PROGRAM pouMachine
VAR
	pnuOn: FB_Motion1way;
	isAirSwitchOn: BOOL;
	tAllPowerOn: BOOL;
	tAnyPowerOn: BOOL;
	tGate1AccessReq: BOOL;
	tGate2AccessReq: BOOL;
	FB_CheckAnyMode_0: FB_CheckAnyMode;
	tWaitMsgXICAdv: BOOL;
	tAnyManualReq: BOOL;
	tAnyAutoReq: BOOL;
END_VAR
VAR // added by the converter: edge detectors and wires of the graphical bodies
    _w1 : BOOL;
END_VAR

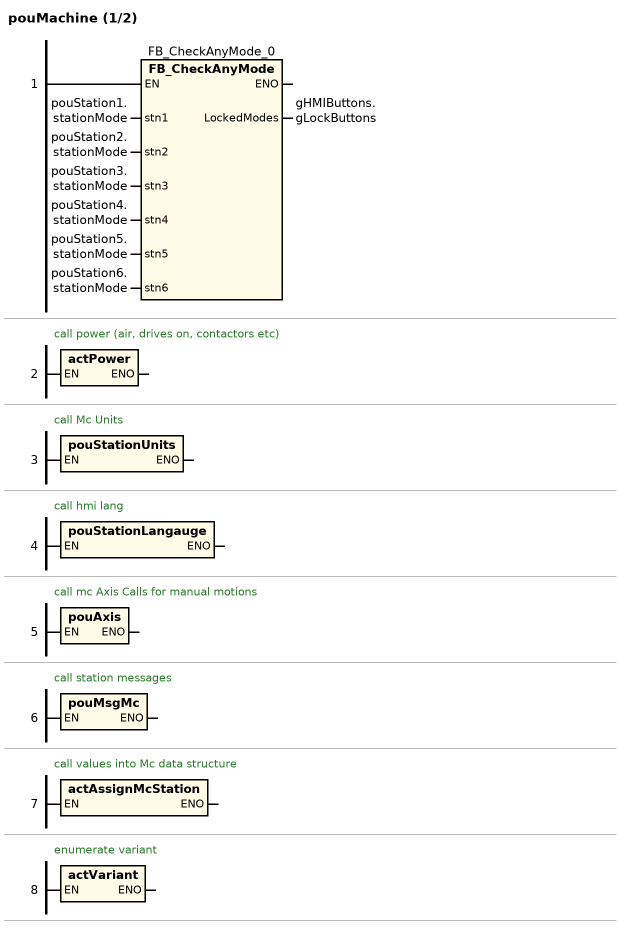
// NETWORK 1
FB_CheckAnyMode_0(
    stn1 := pouStation1.stationMode,
    stn2 := pouStation2.stationMode,
    stn3 := pouStation3.stationMode,
    stn4 := pouStation4.stationMode,
    stn5 := pouStation5.stationMode,
    stn6 := pouStation6.stationMode,
    LockedModes => gHMIButtons.gLockButtons); // FB_CheckAnyMode

// NETWORK 2
// call power (air, drives on, contactors etc)
actPower();

// NETWORK 3
// call Mc Units
pouStationUnits();

// NETWORK 4
// call hmi lang
pouStationLangauge();

// NETWORK 5
// call mc Axis Calls for manual motions
pouAxis();

// NETWORK 6
// call station messages
pouMsgMc();

// NETWORK 7
// call values into Mc data structure
actAssignMcStation();

// NETWORK 8
// enumerate variant
actVariant();

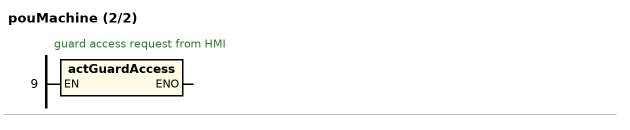
// NETWORK 9
// guard access request from HMI
actGuardAccess();

ACTION actAssignMcStation:
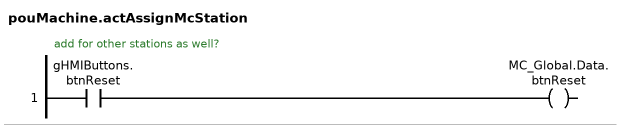
// NETWORK 1
// add for other stations as well?
MC_Global.Data.btnReset := gHMIButtons.btnReset;
END_ACTION

ACTION actGuardAccess:
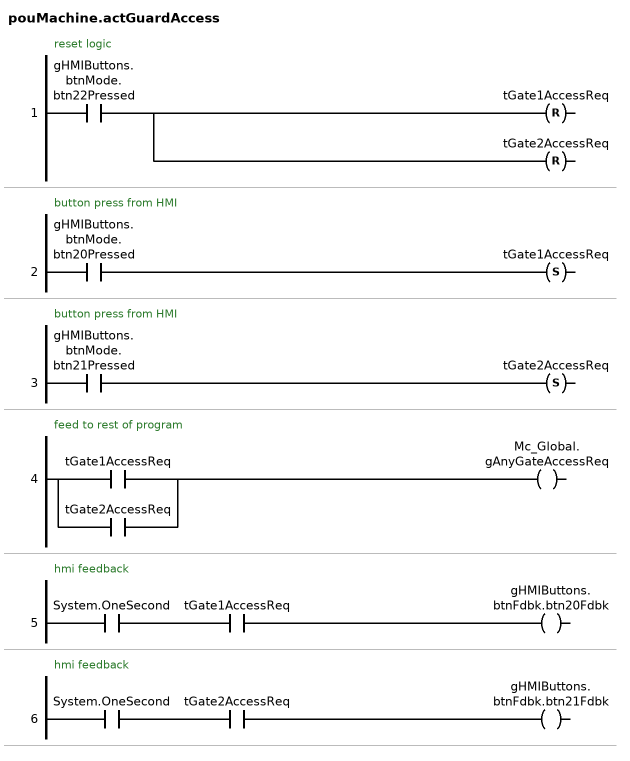
// NETWORK 1
// reset logic
tGate1AccessReq R= gHMIButtons.btnMode.btn22Pressed;
tGate2AccessReq R= gHMIButtons.btnMode.btn22Pressed;

// NETWORK 2
// button press from HMI
tGate1AccessReq S= gHMIButtons.btnMode.btn20Pressed;

// NETWORK 3
// button press from HMI
tGate2AccessReq S= gHMIButtons.btnMode.btn21Pressed;

// NETWORK 4
// feed to rest of program
Mc_Global.gAnyGateAccessReq := tGate1AccessReq OR tGate2AccessReq;

// NETWORK 5
// hmi feedback
gHMIButtons.btnFdbk.btn20Fdbk := System.OneSecond AND tGate1AccessReq;

// NETWORK 6
// hmi feedback
gHMIButtons.btnFdbk.btn21Fdbk := System.OneSecond AND tGate2AccessReq;
END_ACTION

ACTION actPower:
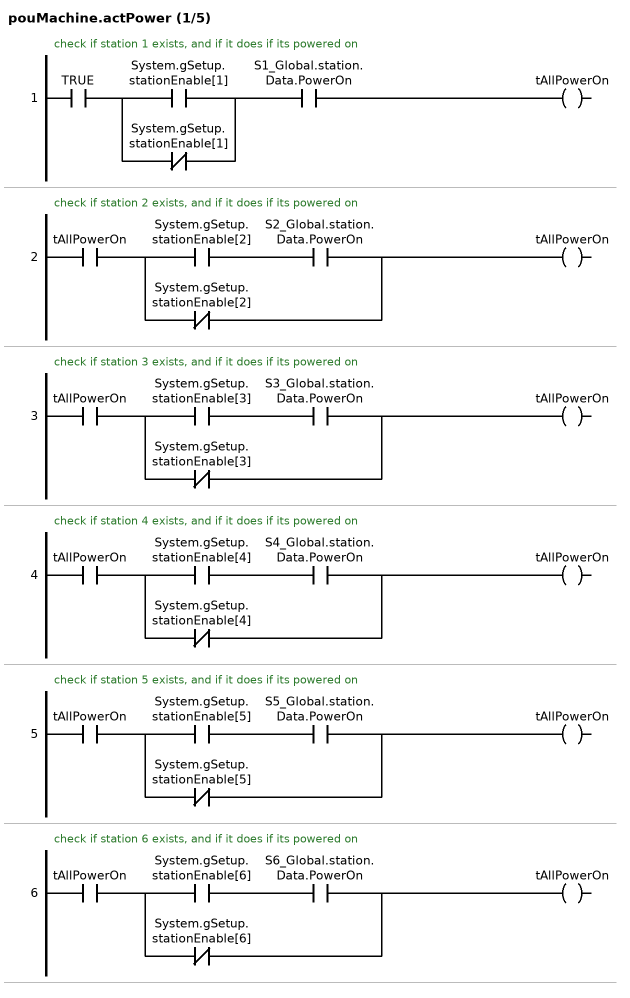
// NETWORK 1
// check if station 1 exists, and if it does if its powered on
tAllPowerOn := TRUE AND (System.gSetup.stationEnable[1] OR NOT System.gSetup.stationEnable[1]) AND S1_Global.station.Data.PowerOn;

// NETWORK 2
// check if station 2 exists, and if it does if its powered on
tAllPowerOn := tAllPowerOn AND (System.gSetup.stationEnable[2] AND S2_Global.station.Data.PowerOn OR NOT System.gSetup.stationEnable[2]);

// NETWORK 3
// check if station 3 exists, and if it does if its powered on
tAllPowerOn := tAllPowerOn AND (System.gSetup.stationEnable[3] AND S3_Global.station.Data.PowerOn OR NOT System.gSetup.stationEnable[3]);

// NETWORK 4
// check if station 4 exists, and if it does if its powered on
tAllPowerOn := tAllPowerOn AND (System.gSetup.stationEnable[4] AND S4_Global.station.Data.PowerOn OR NOT System.gSetup.stationEnable[4]);

// NETWORK 5
// check if station 5 exists, and if it does if its powered on
tAllPowerOn := tAllPowerOn AND (System.gSetup.stationEnable[5] AND S5_Global.station.Data.PowerOn OR NOT System.gSetup.stationEnable[5]);

// NETWORK 6
// check if station 6 exists, and if it does if its powered on
tAllPowerOn := tAllPowerOn AND (System.gSetup.stationEnable[6] AND S6_Global.station.Data.PowerOn OR NOT System.gSetup.stationEnable[6]);

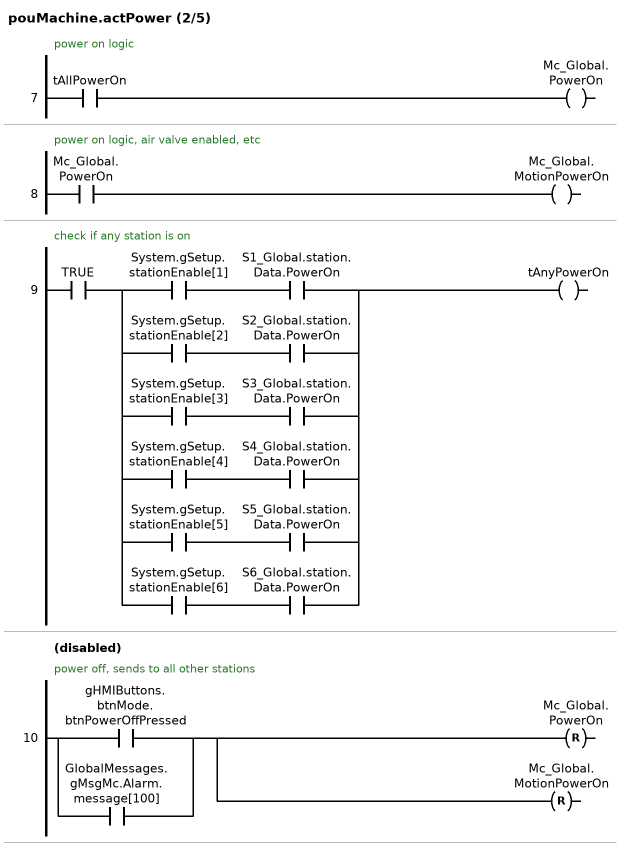
// NETWORK 7
// power on logic
Mc_Global.PowerOn := tAllPowerOn;

// NETWORK 8
// power on logic, air valve enabled, etc
Mc_Global.MotionPowerOn := Mc_Global.PowerOn;

// NETWORK 9
// check if any station is on
tAnyPowerOn := TRUE AND (System.gSetup.stationEnable[1] AND S1_Global.station.Data.PowerOn OR System.gSetup.stationEnable[2] AND S2_Global.station.Data.PowerOn OR System.gSetup.stationEnable[3] AND S3_Global.station.Data.PowerOn OR System.gSetup.stationEnable[4] AND S4_Global.station.Data.PowerOn OR System.gSetup.stationEnable[5] AND S5_Global.station.Data.PowerOn OR System.gSetup.stationEnable[6] AND S6_Global.station.Data.PowerOn);

// NETWORK 10 (disabled)
// power off, sends to all other stations
// _w1 := gHMIButtons.btnMode.btnPowerOffPressed OR GlobalMessages.gMsgMc.Alarm.message[100];
// Mc_Global.PowerOn R= _w1;
// Mc_Global.MotionPowerOn R= _w1;

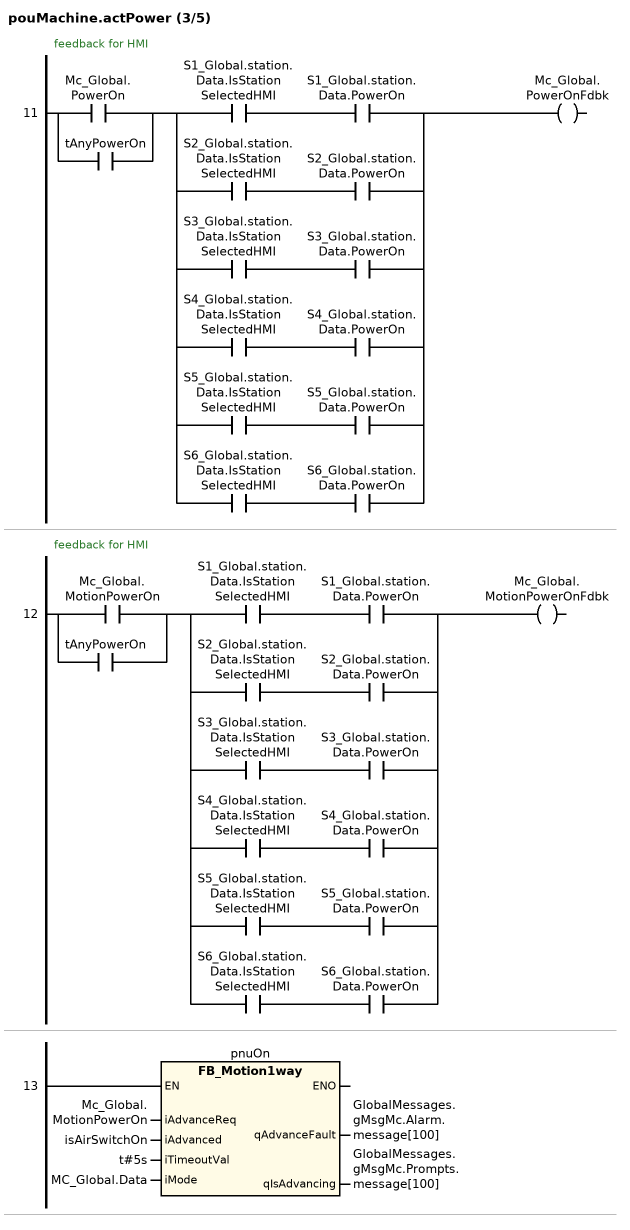
// NETWORK 11
// feedback for HMI
Mc_Global.PowerOnFdbk := (Mc_Global.PowerOn OR tAnyPowerOn) AND (S1_Global.station.Data.IsStationSelectedHMI AND S1_Global.station.Data.PowerOn OR S2_Global.station.Data.IsStationSelectedHMI AND S2_Global.station.Data.PowerOn OR S3_Global.station.Data.IsStationSelectedHMI AND S3_Global.station.Data.PowerOn OR S4_Global.station.Data.IsStationSelectedHMI AND S4_Global.station.Data.PowerOn OR S5_Global.station.Data.IsStationSelectedHMI AND S5_Global.station.Data.PowerOn OR S6_Global.station.Data.IsStationSelectedHMI AND S6_Global.station.Data.PowerOn);

// NETWORK 12
// feedback for HMI
Mc_Global.MotionPowerOnFdbk := (Mc_Global.MotionPowerOn OR tAnyPowerOn) AND (S1_Global.station.Data.IsStationSelectedHMI AND S1_Global.station.Data.PowerOn OR S2_Global.station.Data.IsStationSelectedHMI AND S2_Global.station.Data.PowerOn OR S3_Global.station.Data.IsStationSelectedHMI AND S3_Global.station.Data.PowerOn OR S4_Global.station.Data.IsStationSelectedHMI AND S4_Global.station.Data.PowerOn OR S5_Global.station.Data.IsStationSelectedHMI AND S5_Global.station.Data.PowerOn OR S6_Global.station.Data.IsStationSelectedHMI AND S6_Global.station.Data.PowerOn);

// NETWORK 13
pnuOn(
    iAdvanceReq := Mc_Global.MotionPowerOn,
    iAdvanced := isAirSwitchOn,
    iTimeoutVal := t#5s,
    iMode := MC_Global.Data,
    qAdvanceFault => GlobalMessages.gMsgMc.Alarm.message[100],
    qIsAdvancing => GlobalMessages.gMsgMc.Prompts.message[100]); // FB_Motion1way

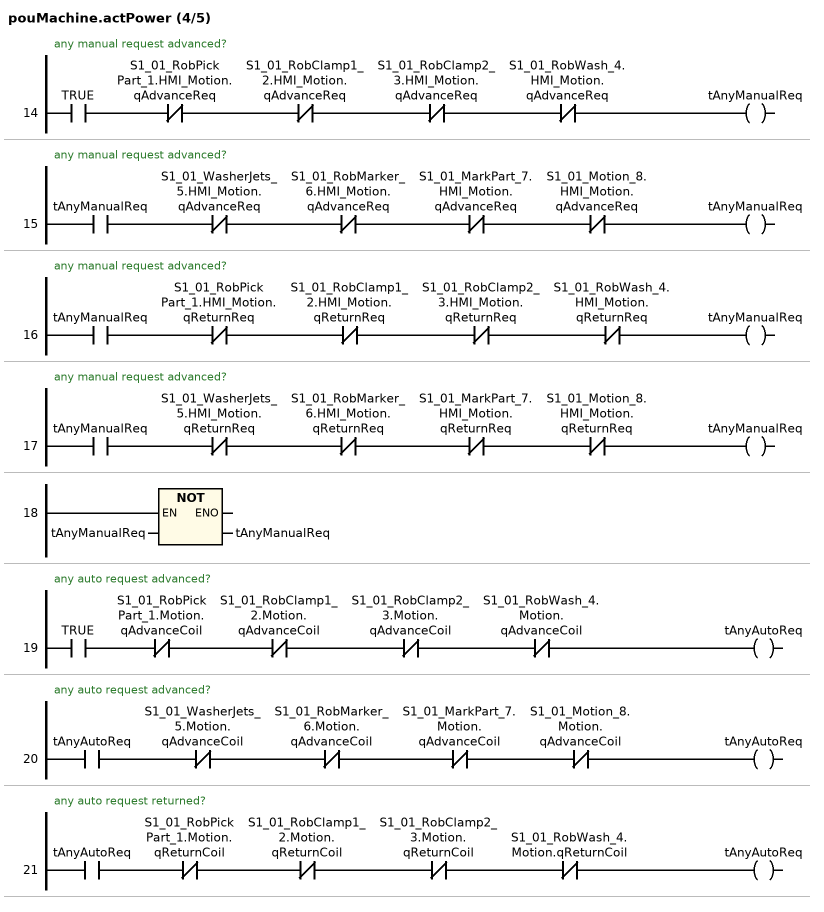
// NETWORK 14
// any manual request advanced?
tAnyManualReq := TRUE AND NOT S1_01_RobPickPart_1.HMI_Motion.qAdvanceReq AND NOT S1_01_RobClamp1_2.HMI_Motion.qAdvanceReq AND NOT S1_01_RobClamp2_3.HMI_Motion.qAdvanceReq AND NOT S1_01_RobWash_4.HMI_Motion.qAdvanceReq;

// NETWORK 15
// any manual request advanced?
tAnyManualReq := tAnyManualReq AND NOT S1_01_WasherJets_5.HMI_Motion.qAdvanceReq AND NOT S1_01_RobMarker_6.HMI_Motion.qAdvanceReq AND NOT S1_01_MarkPart_7.HMI_Motion.qAdvanceReq AND NOT S1_01_Motion_8.HMI_Motion.qAdvanceReq;

// NETWORK 16
// any manual request advanced?
tAnyManualReq := tAnyManualReq AND NOT S1_01_RobPickPart_1.HMI_Motion.qReturnReq AND NOT S1_01_RobClamp1_2.HMI_Motion.qReturnReq AND NOT S1_01_RobClamp2_3.HMI_Motion.qReturnReq AND NOT S1_01_RobWash_4.HMI_Motion.qReturnReq;

// NETWORK 17
// any manual request advanced?
tAnyManualReq := tAnyManualReq AND NOT S1_01_WasherJets_5.HMI_Motion.qReturnReq AND NOT S1_01_RobMarker_6.HMI_Motion.qReturnReq AND NOT S1_01_MarkPart_7.HMI_Motion.qReturnReq AND NOT S1_01_Motion_8.HMI_Motion.qReturnReq;

// NETWORK 18
tAnyManualReq := NOT tAnyManualReq;

// NETWORK 19
// any auto request advanced?
tAnyAutoReq := TRUE AND NOT S1_01_RobPickPart_1.Motion.qAdvanceCoil AND NOT S1_01_RobClamp1_2.Motion.qAdvanceCoil AND NOT S1_01_RobClamp2_3.Motion.qAdvanceCoil AND NOT S1_01_RobWash_4.Motion.qAdvanceCoil;

// NETWORK 20
// any auto request advanced?
tAnyAutoReq := tAnyAutoReq AND NOT S1_01_WasherJets_5.Motion.qAdvanceCoil AND NOT S1_01_RobMarker_6.Motion.qAdvanceCoil AND NOT S1_01_MarkPart_7.Motion.qAdvanceCoil AND NOT S1_01_Motion_8.Motion.qAdvanceCoil;

// NETWORK 21
// any auto request returned?
tAnyAutoReq := tAnyAutoReq AND NOT S1_01_RobPickPart_1.Motion.qReturnCoil AND NOT S1_01_RobClamp1_2.Motion.qReturnCoil AND NOT S1_01_RobClamp2_3.Motion.qReturnCoil AND NOT S1_01_RobWash_4.Motion.qReturnCoil;

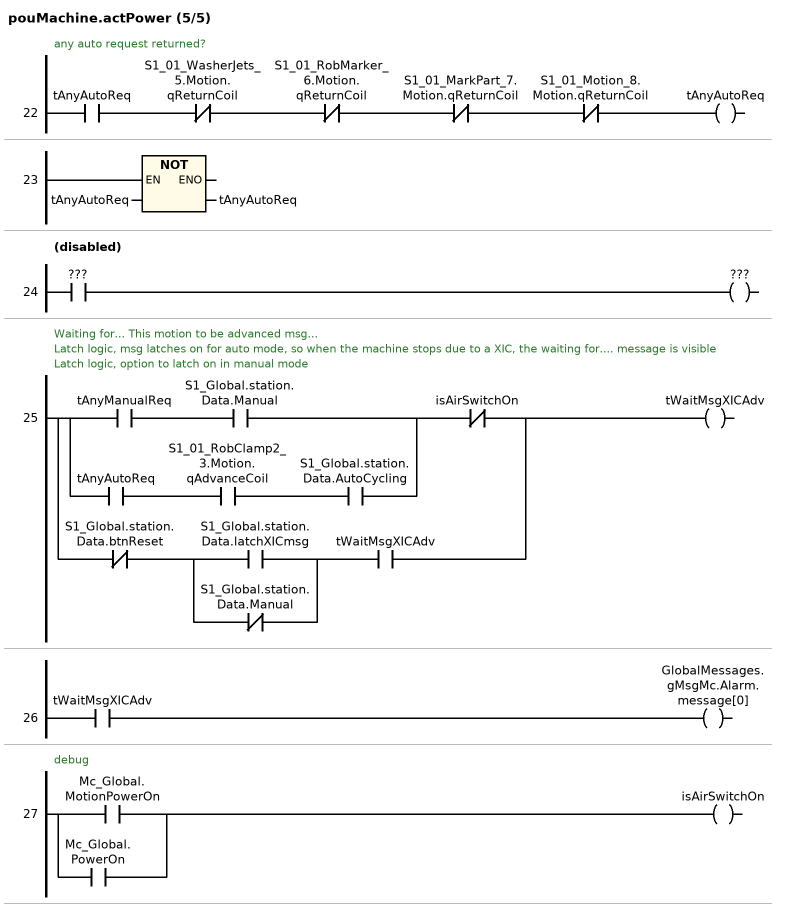
// NETWORK 22
// any auto request returned?
tAnyAutoReq := tAnyAutoReq AND NOT S1_01_WasherJets_5.Motion.qReturnCoil AND NOT S1_01_RobMarker_6.Motion.qReturnCoil AND NOT S1_01_MarkPart_7.Motion.qReturnCoil AND NOT S1_01_Motion_8.Motion.qReturnCoil;

// NETWORK 23
tAnyAutoReq := NOT tAnyAutoReq;

// NETWORK 24 (disabled)
// ??? := ???;

// NETWORK 25
// Waiting for... This motion to be advanced msg...
// Latch logic, msg latches on for auto mode, so when the machine stops due to a XIC, the waiting for.... message is visible
// Latch logic, option to latch on in manual mode
tWaitMsgXICAdv := (tAnyManualReq AND S1_Global.station.Data.Manual OR tAnyAutoReq AND S1_01_RobClamp2_3.Motion.qAdvanceCoil AND S1_Global.station.Data.AutoCycling) AND NOT isAirSwitchOn OR NOT S1_Global.station.Data.btnReset AND (S1_Global.station.Data.latchXICmsg OR NOT S1_Global.station.Data.Manual) AND tWaitMsgXICAdv;

// NETWORK 26
GlobalMessages.gMsgMc.Alarm.message[0] := tWaitMsgXICAdv;

// NETWORK 27
// debug
isAirSwitchOn := Mc_Global.MotionPowerOn OR Mc_Global.PowerOn;
END_ACTION

ACTION actVariant:
//clear down variant
//Mc_Variant.gVariantSelected	:= 2#00000000000000000000000000000000;

//insert into control DWORD to clear down future memory allocations
{IF defined (NoPLC)}
    Mc_Variant.gVariantSelected	:= 2#00000000000000000000000000000001;
{ELSIF defined (PLCTest)}
 	Mc_Variant.gVariantSelected	:= 2#00000000000000000000000000000010;
{END_IF}

//with the DWORD cleared down, then enumerate the variant
IF Mc_Variant.gVariantSelected = 2#00000000000000000000000000000001 THEN 	Mc_Variant.gIsNoPLC		:= TRUE; ELSE Mc_Variant.gIsNoPLC		:= FALSE; END_IF
IF Mc_Variant.gVariantSelected = 2#00000000000000000000000000000010 THEN	Mc_Variant.gIsPLCTest	:= TRUE; ELSE Mc_Variant.gIsPLCTest		:= FALSE; END_IF
IF Mc_Variant.gVariantSelected = 2#00000000000000000000000000000110 THEN	Mc_Variant.gIsVariant1	:= TRUE; ELSE Mc_Variant.gIsVariant1	:= FALSE; END_IF
IF Mc_Variant.gVariantSelected = 2#00000000000000000000000000001000 THEN	Mc_Variant.gIsVariant2	:= TRUE; ELSE Mc_Variant.gIsVariant2	:= FALSE; END_IF
IF Mc_Variant.gVariantSelected = 2#00000000000000000000000000010000 THEN	Mc_Variant.gIsVariant3	:= TRUE; ELSE Mc_Variant.gIsVariant3	:= FALSE; END_IF
IF Mc_Variant.gVariantSelected = 2#00000000000000000000000000100000 THEN	Mc_Variant.gIsVariant4	:= TRUE; ELSE Mc_Variant.gIsVariant4	:= FALSE; END_IF
IF Mc_Variant.gVariantSelected = 2#00000000000000000000000001000000 THEN	Mc_Variant.gIsVariant5	:= TRUE; ELSE Mc_Variant.gIsVariant5	:= FALSE; END_IF
IF Mc_Variant.gVariantSelected = 2#00000000000000000000000010000000 THEN	Mc_Variant.gIsVariant6	:= TRUE; ELSE Mc_Variant.gIsVariant6	:= FALSE; END_IF
IF Mc_Variant.gVariantSelected = 2#00000000000000000000000100000000 THEN	Mc_Variant.gIsVariant7	:= TRUE; ELSE Mc_Variant.gIsVariant7	:= FALSE; END_IF
//etc
END_ACTION

END_PROGRAM

(* stored: Version 1.1.0.1, ProductVersion 3.1.4024.11
   POU pouMachine: Id {130f38d3-d0ad-451a-83e5-25f291f23105}, SpecialFunc None
   Action actAssignMcStation: Id {86f27bdf-cbff-4efe-a514-d6c2d712b080}
   Action actGuardAccess: Id {d0c105ec-7d4a-0556-3deb-638d3ce8d5f1}
   Action actPower: Id {2ab649fa-87ba-4e15-a599-af17da8737b9}
   Action actVariant: Id {a6d5b483-94b7-4903-8313-6221ffbc9d3f} *)
